(* Logix 5000 project; controller TEC_81 vendor 1 type 14 code 148 rev 36.11; software revision 36.00; part 2 of 4 *)
(* tags used below, declared in another part *)
   Axis_1 : AXIS_CIP_DRIVE;
   Axis_2 : AXIS_CIP_DRIVE;   // Almacen 2
   B_Reset_Posicion_kinetix : DINT;
   Ctrl_Kinetix_A2 : DINT;   // Boton Start Kinetix
   DestornilladorEnPosicion_Mesa : BOOL;   // Sensor de posición de Destornillador en Mesa Central
   Done_Kinetx : DINT;
   Extender_Piston_1_Mesa_Kuka : BOOL;   // Extender Pistón Esquina de Mesa Central
   Extender_Piston_2_Mesa_Kuka : BOOL;   // Extender Pistón Centro de Mesa Central
   Faul_Axis : DINT;
   GripperEnPosicion_Mesa : BOOL;   // Sensor de posición de Gripper en Mesa Central
   In_Pos_Alm_1 : DINT;
   In_Pos_Alm_2 : DINT;
   Kinetix_Pos_Alm_1 : DINT;
   Kinetix_Pos_Alm_2 : DINT;
   KUKA : TIMER;
   MAFR_Mtr_Alm_1 : MOTION_INSTRUCTION;
   MAFR_Mtr_Alm_2 : MOTION_INSTRUCTION;
   MAM_1_Mtr_Alm_0 : MOTION_INSTRUCTION;
   MAM_1_Mtr_Alm_1 : MOTION_INSTRUCTION;
   MAM_1_Mtr_Alm_2 : MOTION_INSTRUCTION;
   MAM_2_Mtr_Alm_1 : MOTION_INSTRUCTION;
   MAM_2_Mtr_Alm_2 : MOTION_INSTRUCTION;
   MAM_3_Mtr_Alm_1 : MOTION_INSTRUCTION;
   MAM_3_Mtr_Alm_2 : MOTION_INSTRUCTION;
   MAM_4_Mtr_Alm_1 : MOTION_INSTRUCTION;
   MAM_4_Mtr_Alm_2 : MOTION_INSTRUCTION;
   MAM_5_Mtr_Alm_1 : MOTION_INSTRUCTION;
   MAM_5_Mtr_Alm_2 : MOTION_INSTRUCTION;
   MAM_6_Mtr_Alm_2 : MOTION_INSTRUCTION;
   ok_com : BOOL;   // tag de prueba de comunicacion
   reset_Kinetix : BOOL;
   Retraer_Piston_1_Mesa_Kuka : BOOL;   // Retraer Pistón Esquina de Mesa Central
   Retraer_Piston_2_Mesa_Kuka : BOOL;   // Retraer Pistón Centro de Mesa Central
   Sensor_Piston_1_Ext_Mesa : BOOL;   // Sensor de Piston Extendido Esquina de la Mesa Central
   Sensor_Piston_1_Ret_Mesa : BOOL;   // Sensor de Pistón Retraido Esquina de la Mesa Central
   Sensor_Piston_2_Ext_Mesa : BOOL;   // Sensor de Pistón Extendido Centro de la Mesa Central
   Sensor_Piston_2_Ret_Mesa : BOOL;   // Sensor de Pistón Retraido Centro de la Mesa Central
   servo_start : MOTION_INSTRUCTION;
   servo_start_01 : MOTION_INSTRUCTION;
   Sevo_Stop : MOTION_INSTRUCTION;
   Start_Kinetix_Alm_1 : DINT;
   Start_Kinetix_Alm_2 : DINT;
   Test : BOOL;
   To_Pos_Alm_1 : DINT;
   To_Pos_Alm_2 : DINT;
   VentosaEnPosicion_Mesa : BOOL;   // Sensor de posición de Ventosa en Mesa Central

PROGRAM _05_Mesa_Central   (* main routine _01_Main *)

ROUTINE _01_Main   (* ladder *)
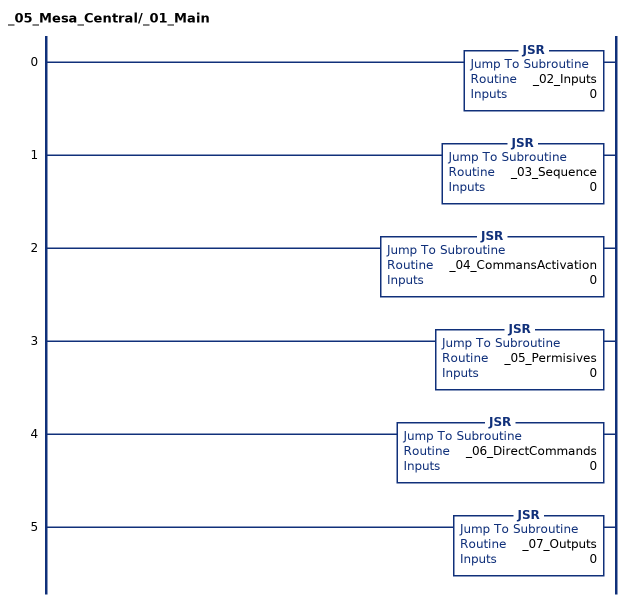
   0: JSR(_02_Inputs,0);
   1: JSR(_03_Sequence,0);
   2: JSR(_04_CommansActivation,0);
   3: JSR(_05_Permisives,0);
   4: JSR(_06_DirectCommands,0);
   5: JSR(_07_Outputs,0);
END_ROUTINE

ROUTINE _02_Inputs   (* ladder *)
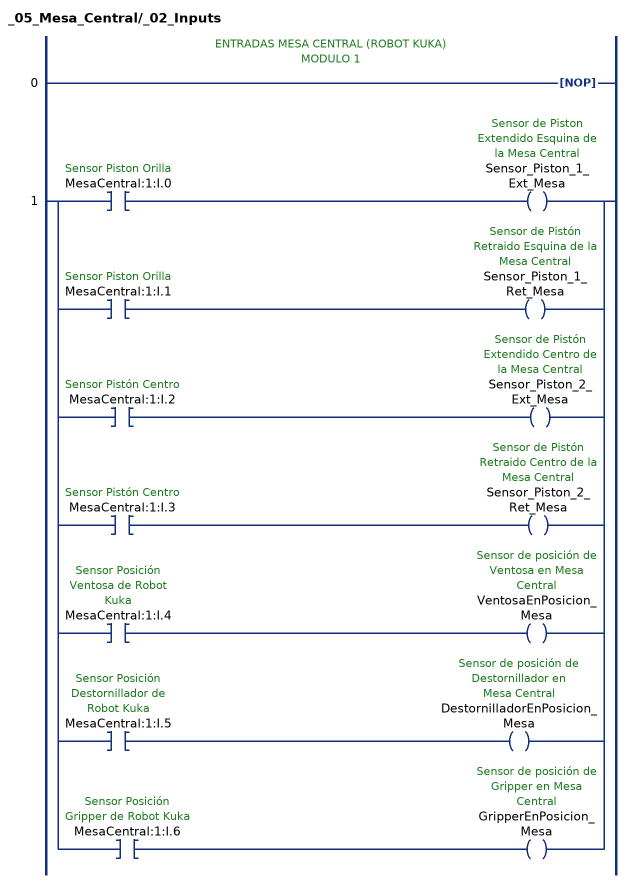
   // ENTRADAS MESA CENTRAL (ROBOT KUKA)
   // MODULO 1
   0: NOP();
   1: [XIC(MesaCentral:1:I.0) OTE(Sensor_Piston_1_Ext_Mesa) ,XIC(MesaCentral:1:I.1) OTE(Sensor_Piston_1_Ret_Mesa) ,XIC(MesaCentral:1:I.2) OTE(Sensor_Piston_2_Ext_Mesa) ,XIC(MesaCentral:1:I.3) OTE(Sensor_Piston_2_Ret_Mesa) ,XIC(MesaCentral:1:I.4) OTE(VentosaEnPosicion_Mesa) ,XIC(MesaCentral:1:I.5) OTE(DestornilladorEnPosicion_Mesa) ,XIC(MesaCentral:1:I.6) OTE(GripperEnPosicion_Mesa) ];
END_ROUTINE

ROUTINE _03_Sequence   (* ladder *)
END_ROUTINE

ROUTINE _04_CommansActivation   (* ladder *)
END_ROUTINE

ROUTINE _05_Permisives   (* ladder *)
END_ROUTINE

ROUTINE _06_DirectCommands   (* ladder *)
END_ROUTINE

ROUTINE _07_Outputs   (* ladder *)
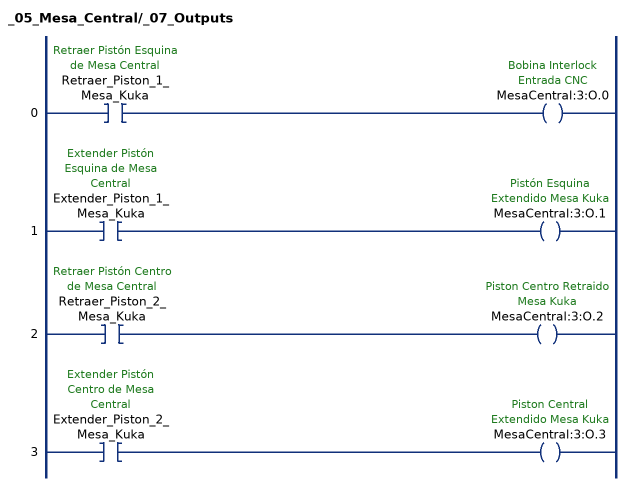
   0: XIC(Retraer_Piston_1_Mesa_Kuka)OTE(MesaCentral:3:O.0);
   1: XIC(Extender_Piston_1_Mesa_Kuka)OTE(MesaCentral:3:O.1);
   2: XIC(Retraer_Piston_2_Mesa_Kuka)OTE(MesaCentral:3:O.2);
   3: XIC(Extender_Piston_2_Mesa_Kuka)OTE(MesaCentral:3:O.3);
END_ROUTINE

ROUTINE test   (* sequential function chart *)
END_ROUTINE

ROUTINE test1   (* ladder *)
END_ROUTINE
END_PROGRAM

PROGRAM _Almacen_1   (* main routine _01_Main_Alm_11 *)
VAR
   B_Reset_Posicion_kinetix_0 : DINT;
   Ctrl_Kinetix_A1 : DINT;
   Done_Kinetx_0 : DINT;
   home_step_1 : BOOL;
   Kinetix_Pos_Alm_0 : DINT;
   ok_com_1 : BOOL;
   reset_Kinetix_1 : BOOL;
END_VAR

ROUTINE _01_Main_Alm_11   (* ladder *)
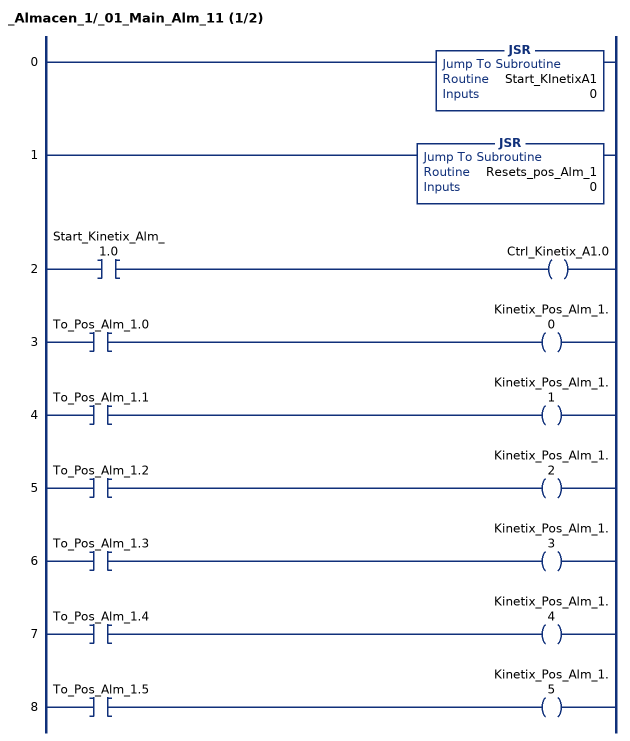
   0: JSR(Start_KInetixA1,0);
   1: JSR(Resets_pos_Alm_1,0);
   2: XIC(Start_Kinetix_Alm_1.0)OTE(Ctrl_Kinetix_A1.0);
   3: XIC(To_Pos_Alm_1.0)OTE(Kinetix_Pos_Alm_1.0);
   4: XIC(To_Pos_Alm_1.1)OTE(Kinetix_Pos_Alm_1.1);
   5: XIC(To_Pos_Alm_1.2)OTE(Kinetix_Pos_Alm_1.2);
   6: XIC(To_Pos_Alm_1.3)OTE(Kinetix_Pos_Alm_1.3);
   7: XIC(To_Pos_Alm_1.4)OTE(Kinetix_Pos_Alm_1.4);
   8: XIC(To_Pos_Alm_1.5)OTE(Kinetix_Pos_Alm_1.5);
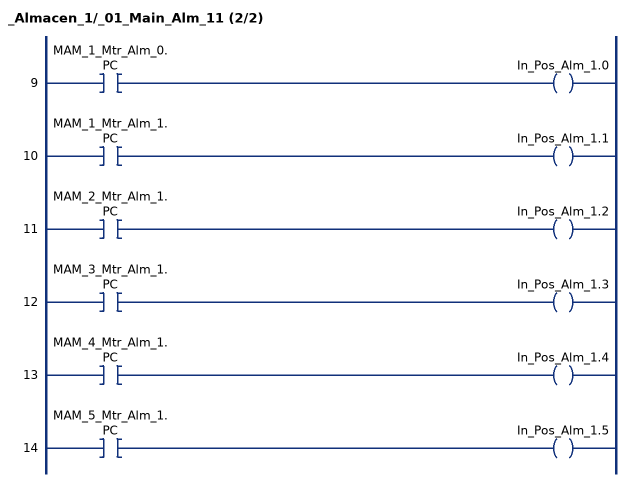
   9: XIC(MAM_1_Mtr_Alm_0.PC)OTE(In_Pos_Alm_1.0);
   10: XIC(MAM_1_Mtr_Alm_1.PC)OTE(In_Pos_Alm_1.1);
   11: XIC(MAM_2_Mtr_Alm_1.PC)OTE(In_Pos_Alm_1.2);
   12: XIC(MAM_3_Mtr_Alm_1.PC)OTE(In_Pos_Alm_1.3);
   13: XIC(MAM_4_Mtr_Alm_1.PC)OTE(In_Pos_Alm_1.4);
   14: XIC(MAM_5_Mtr_Alm_1.PC)OTE(In_Pos_Alm_1.5);
END_ROUTINE

ROUTINE Resets_pos_Alm_1   (* ladder *)
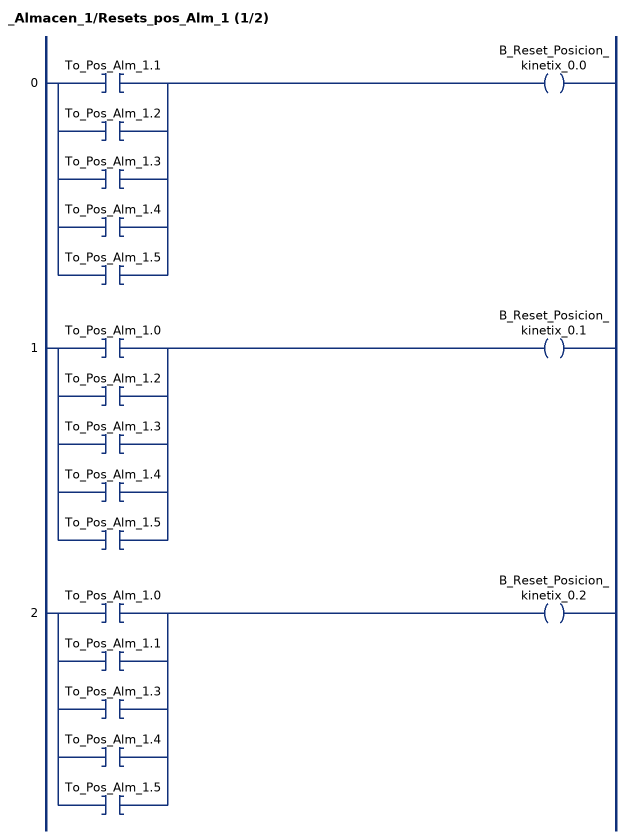
   0: [XIC(To_Pos_Alm_1.1) ,XIC(To_Pos_Alm_1.2) ,XIC(To_Pos_Alm_1.3) ,XIC(To_Pos_Alm_1.4) ,XIC(To_Pos_Alm_1.5) ]OTE(B_Reset_Posicion_kinetix_0.0);
   1: [XIC(To_Pos_Alm_1.0) ,XIC(To_Pos_Alm_1.2) ,XIC(To_Pos_Alm_1.3) ,XIC(To_Pos_Alm_1.4) ,XIC(To_Pos_Alm_1.5) ]OTE(B_Reset_Posicion_kinetix_0.1);
   2: [XIC(To_Pos_Alm_1.0) ,XIC(To_Pos_Alm_1.1) ,XIC(To_Pos_Alm_1.3) ,XIC(To_Pos_Alm_1.4) ,XIC(To_Pos_Alm_1.5) ]OTE(B_Reset_Posicion_kinetix_0.2);
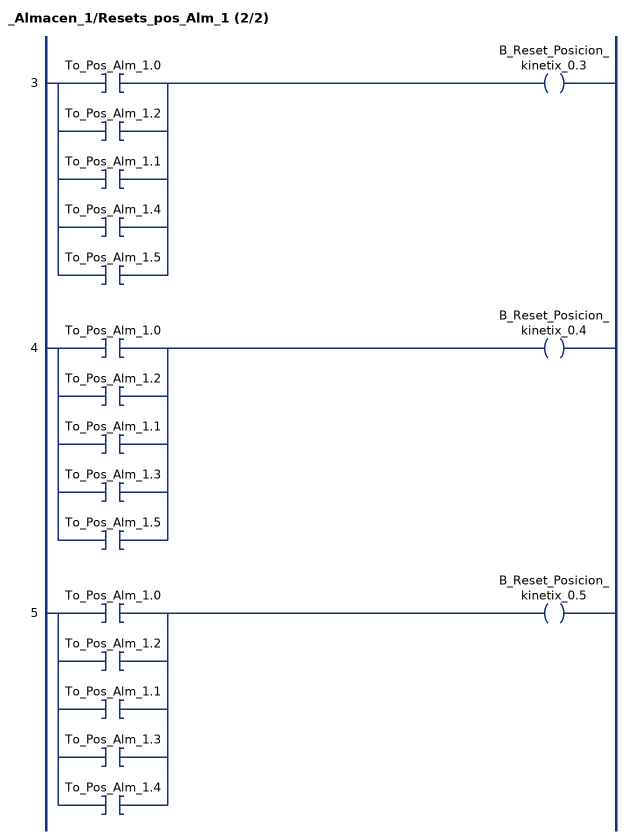
   3: [XIC(To_Pos_Alm_1.0) ,XIC(To_Pos_Alm_1.2) ,XIC(To_Pos_Alm_1.1) ,XIC(To_Pos_Alm_1.4) ,XIC(To_Pos_Alm_1.5) ]OTE(B_Reset_Posicion_kinetix_0.3);
   4: [XIC(To_Pos_Alm_1.0) ,XIC(To_Pos_Alm_1.2) ,XIC(To_Pos_Alm_1.1) ,XIC(To_Pos_Alm_1.3) ,XIC(To_Pos_Alm_1.5) ]OTE(B_Reset_Posicion_kinetix_0.4);
   5: [XIC(To_Pos_Alm_1.0) ,XIC(To_Pos_Alm_1.2) ,XIC(To_Pos_Alm_1.1) ,XIC(To_Pos_Alm_1.3) ,XIC(To_Pos_Alm_1.4) ]OTE(B_Reset_Posicion_kinetix_0.5);
END_ROUTINE

ROUTINE Start_KInetixA1   (* ladder *)
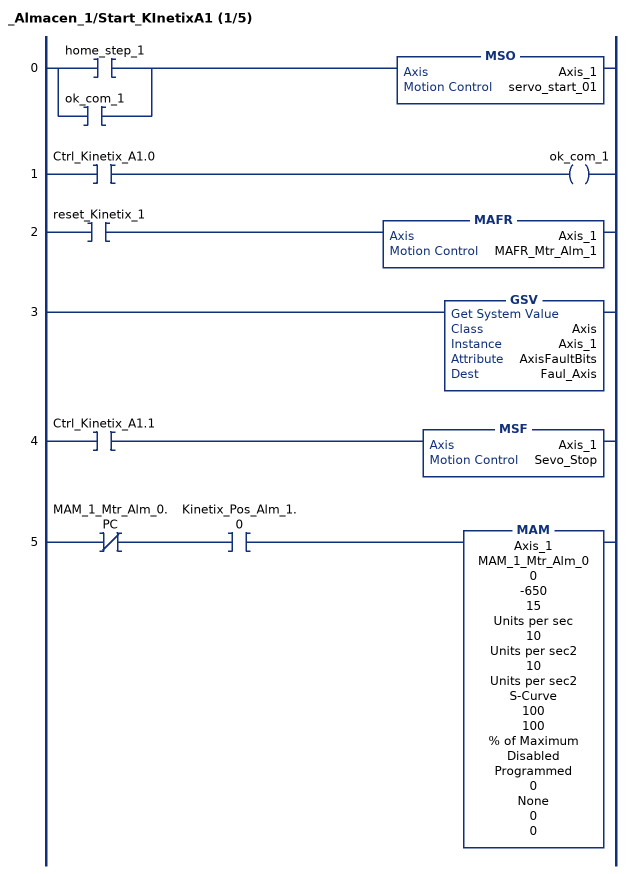
   0: [XIC(home_step_1) ,XIC(ok_com_1) ]MSO(Axis_1,servo_start_01);
   1: XIC(Ctrl_Kinetix_A1.0)OTE(ok_com_1);
   2: XIC(reset_Kinetix_1)MAFR(Axis_1,MAFR_Mtr_Alm_1);
   3: GSV(Axis,Axis_1,AxisFaultBits,Faul_Axis);
   4: XIC(Ctrl_Kinetix_A1.1)MSF(Axis_1,Sevo_Stop);
   5: XIO(MAM_1_Mtr_Alm_0.PC)XIC(Kinetix_Pos_Alm_1.0)MAM(Axis_1,MAM_1_Mtr_Alm_0,0,-650,15,Units per sec,10,Units per sec2,10,Units per sec2,S-Curve,100,100,% of Maximum,Disabled,Programmed,0,None,0,0);
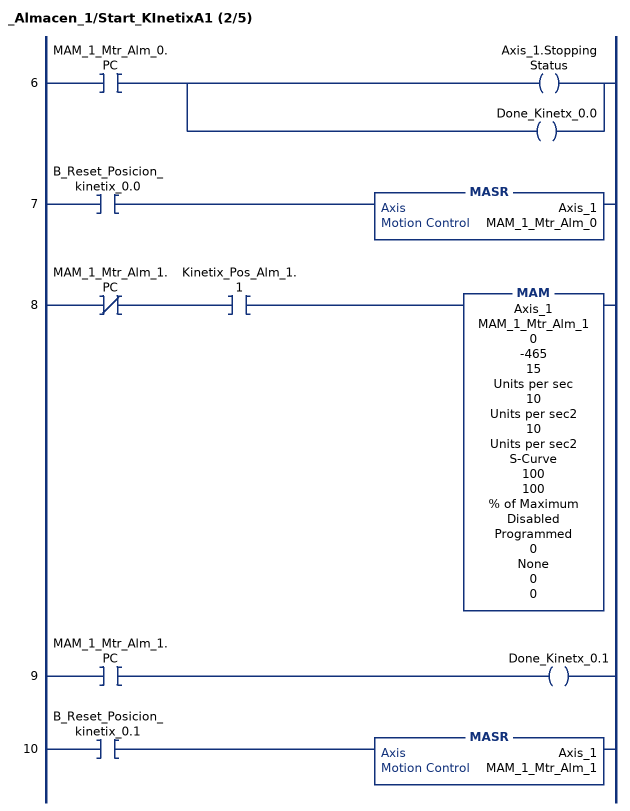
   6: XIC(MAM_1_Mtr_Alm_0.PC)[OTE(Axis_1.StoppingStatus) ,OTE(Done_Kinetx_0.0) ];
   7: XIC(B_Reset_Posicion_kinetix_0.0)MASR(Axis_1,MAM_1_Mtr_Alm_0);
   8: XIO(MAM_1_Mtr_Alm_1.PC)XIC(Kinetix_Pos_Alm_1.1)MAM(Axis_1,MAM_1_Mtr_Alm_1,0,-465,15,Units per sec,10,Units per sec2,10,Units per sec2,S-Curve,100,100,% of Maximum,Disabled,Programmed,0,None,0,0);
   9: XIC(MAM_1_Mtr_Alm_1.PC)OTE(Done_Kinetx_0.1);
   10: XIC(B_Reset_Posicion_kinetix_0.1)MASR(Axis_1,MAM_1_Mtr_Alm_1);
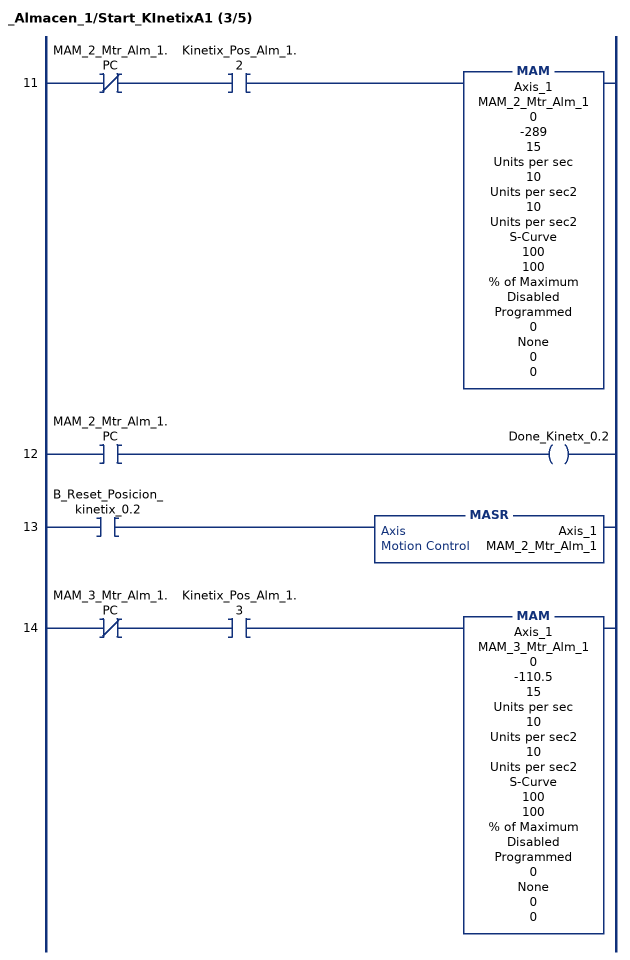
   11: XIO(MAM_2_Mtr_Alm_1.PC)XIC(Kinetix_Pos_Alm_1.2)MAM(Axis_1,MAM_2_Mtr_Alm_1,0,-289,15,Units per sec,10,Units per sec2,10,Units per sec2,S-Curve,100,100,% of Maximum,Disabled,Programmed,0,None,0,0);
   12: XIC(MAM_2_Mtr_Alm_1.PC)OTE(Done_Kinetx_0.2);
   13: XIC(B_Reset_Posicion_kinetix_0.2)MASR(Axis_1,MAM_2_Mtr_Alm_1);
   14: XIO(MAM_3_Mtr_Alm_1.PC)XIC(Kinetix_Pos_Alm_1.3)MAM(Axis_1,MAM_3_Mtr_Alm_1,0,-110.5,15,Units per sec,10,Units per sec2,10,Units per sec2,S-Curve,100,100,% of Maximum,Disabled,Programmed,0,None,0,0);
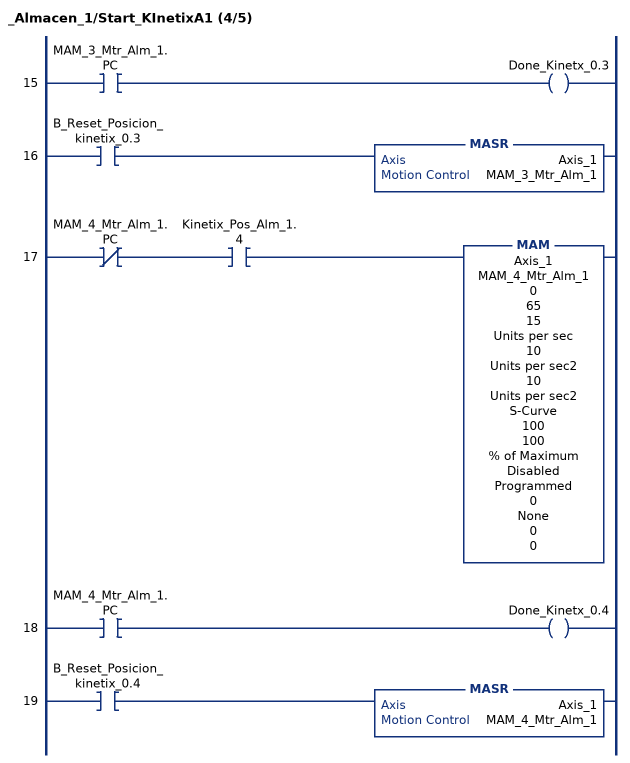
   15: XIC(MAM_3_Mtr_Alm_1.PC)OTE(Done_Kinetx_0.3);
   16: XIC(B_Reset_Posicion_kinetix_0.3)MASR(Axis_1,MAM_3_Mtr_Alm_1);
   17: XIO(MAM_4_Mtr_Alm_1.PC)XIC(Kinetix_Pos_Alm_1.4)MAM(Axis_1,MAM_4_Mtr_Alm_1,0,65,15,Units per sec,10,Units per sec2,10,Units per sec2,S-Curve,100,100,% of Maximum,Disabled,Programmed,0,None,0,0);
   18: XIC(MAM_4_Mtr_Alm_1.PC)OTE(Done_Kinetx_0.4);
   19: XIC(B_Reset_Posicion_kinetix_0.4)MASR(Axis_1,MAM_4_Mtr_Alm_1);
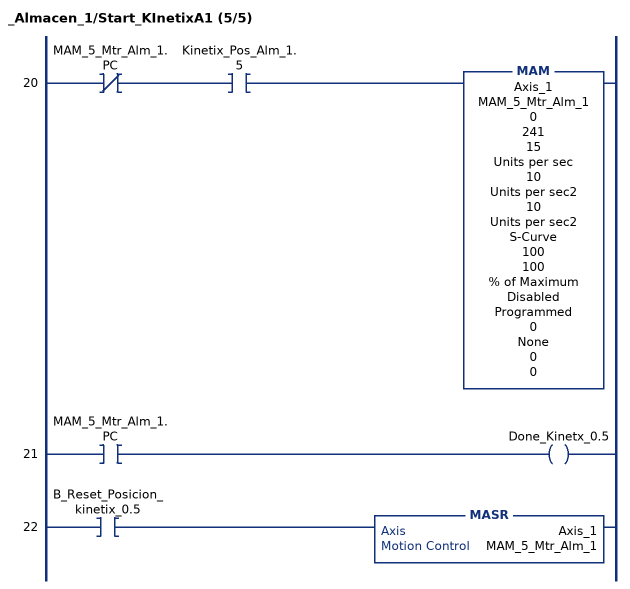
   20: XIO(MAM_5_Mtr_Alm_1.PC)XIC(Kinetix_Pos_Alm_1.5)MAM(Axis_1,MAM_5_Mtr_Alm_1,0,241,15,Units per sec,10,Units per sec2,10,Units per sec2,S-Curve,100,100,% of Maximum,Disabled,Programmed,0,None,0,0);
   21: XIC(MAM_5_Mtr_Alm_1.PC)OTE(Done_Kinetx_0.5);
   22: XIC(B_Reset_Posicion_kinetix_0.5)MASR(Axis_1,MAM_5_Mtr_Alm_1);
END_ROUTINE
END_PROGRAM

PROGRAM _Almacen_2   (* main routine _01_Main *)
VAR
   home_step : BOOL;
END_VAR

ROUTINE _01_Main   (* ladder *)
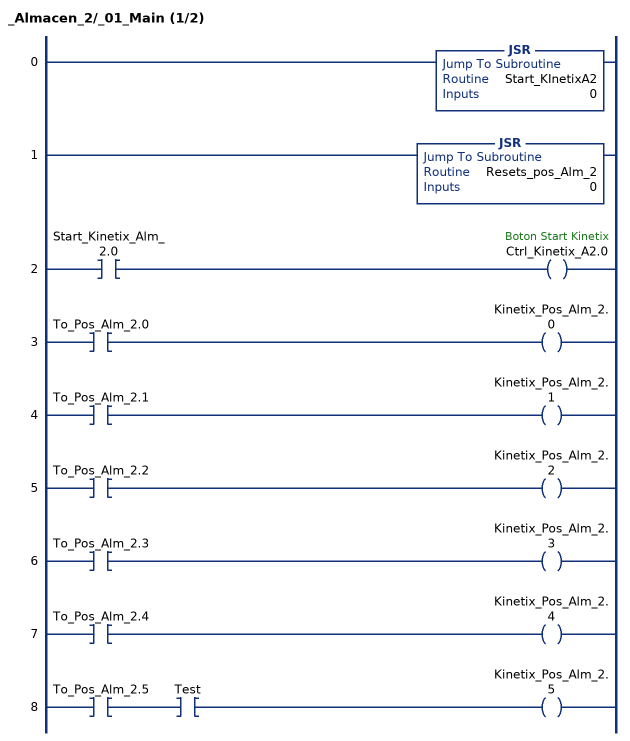
   0: JSR(Start_KInetixA2,0);
   1: JSR(Resets_pos_Alm_2,0);
   2: XIC(Start_Kinetix_Alm_2.0)OTE(Ctrl_Kinetix_A2.0);
   3: XIC(To_Pos_Alm_2.0)OTE(Kinetix_Pos_Alm_2.0);
   4: XIC(To_Pos_Alm_2.1)OTE(Kinetix_Pos_Alm_2.1);
   5: XIC(To_Pos_Alm_2.2)OTE(Kinetix_Pos_Alm_2.2);
   6: XIC(To_Pos_Alm_2.3)OTE(Kinetix_Pos_Alm_2.3);
   7: XIC(To_Pos_Alm_2.4)OTE(Kinetix_Pos_Alm_2.4);
   8: XIC(To_Pos_Alm_2.5)XIC(Test)OTE(Kinetix_Pos_Alm_2.5);
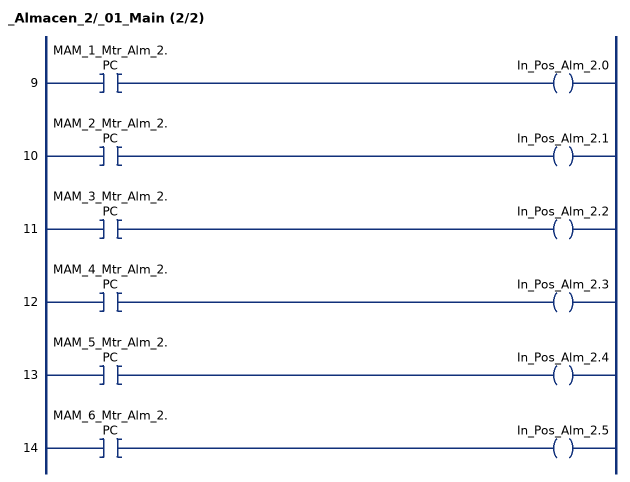
   9: XIC(MAM_1_Mtr_Alm_2.PC)OTE(In_Pos_Alm_2.0);
   10: XIC(MAM_2_Mtr_Alm_2.PC)OTE(In_Pos_Alm_2.1);
   11: XIC(MAM_3_Mtr_Alm_2.PC)OTE(In_Pos_Alm_2.2);
   12: XIC(MAM_4_Mtr_Alm_2.PC)OTE(In_Pos_Alm_2.3);
   13: XIC(MAM_5_Mtr_Alm_2.PC)OTE(In_Pos_Alm_2.4);
   14: XIC(MAM_6_Mtr_Alm_2.PC)OTE(In_Pos_Alm_2.5);
END_ROUTINE

ROUTINE Resets_pos_Alm_2   (* ladder *)
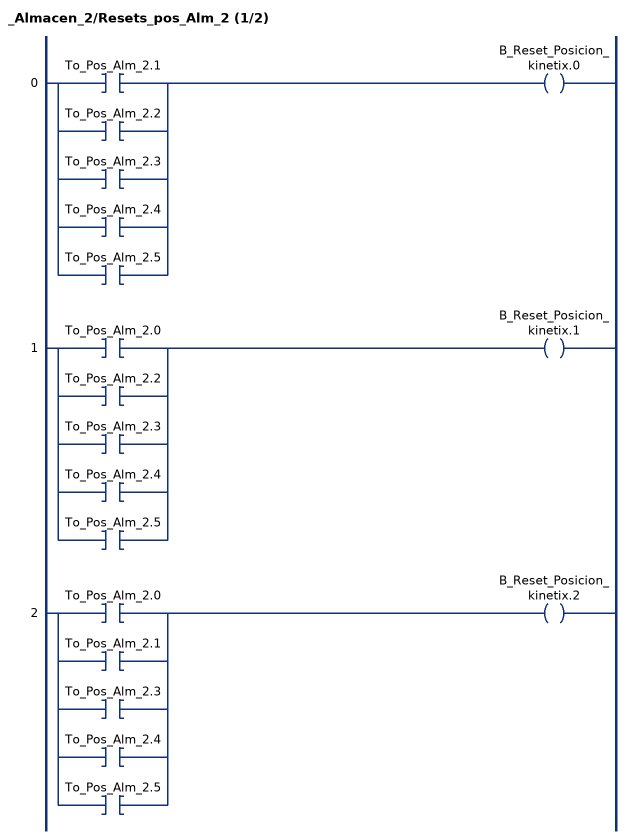
   0: [XIC(To_Pos_Alm_2.1) ,XIC(To_Pos_Alm_2.2) ,XIC(To_Pos_Alm_2.3) ,XIC(To_Pos_Alm_2.4) ,XIC(To_Pos_Alm_2.5) ]OTE(B_Reset_Posicion_kinetix.0);
   1: [XIC(To_Pos_Alm_2.0) ,XIC(To_Pos_Alm_2.2) ,XIC(To_Pos_Alm_2.3) ,XIC(To_Pos_Alm_2.4) ,XIC(To_Pos_Alm_2.5) ]OTE(B_Reset_Posicion_kinetix.1);
   2: [XIC(To_Pos_Alm_2.0) ,XIC(To_Pos_Alm_2.1) ,XIC(To_Pos_Alm_2.3) ,XIC(To_Pos_Alm_2.4) ,XIC(To_Pos_Alm_2.5) ]OTE(B_Reset_Posicion_kinetix.2);
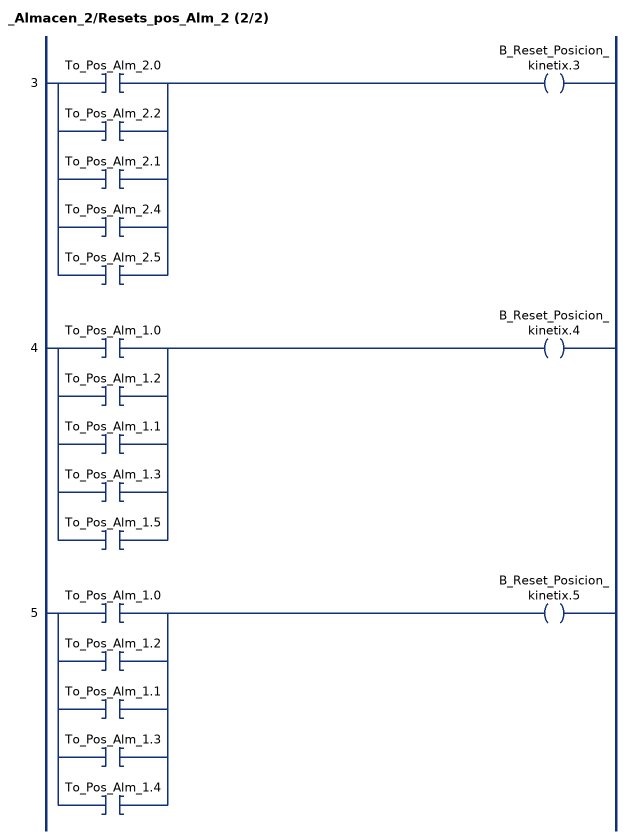
   3: [XIC(To_Pos_Alm_2.0) ,XIC(To_Pos_Alm_2.2) ,XIC(To_Pos_Alm_2.1) ,XIC(To_Pos_Alm_2.4) ,XIC(To_Pos_Alm_2.5) ]OTE(B_Reset_Posicion_kinetix.3);
   4: [XIC(To_Pos_Alm_1.0) ,XIC(To_Pos_Alm_1.2) ,XIC(To_Pos_Alm_1.1) ,XIC(To_Pos_Alm_1.3) ,XIC(To_Pos_Alm_1.5) ]OTE(B_Reset_Posicion_kinetix.4);
   5: [XIC(To_Pos_Alm_1.0) ,XIC(To_Pos_Alm_1.2) ,XIC(To_Pos_Alm_1.1) ,XIC(To_Pos_Alm_1.3) ,XIC(To_Pos_Alm_1.4) ]OTE(B_Reset_Posicion_kinetix.5);
END_ROUTINE

ROUTINE Start_KInetixA2   (* ladder *)
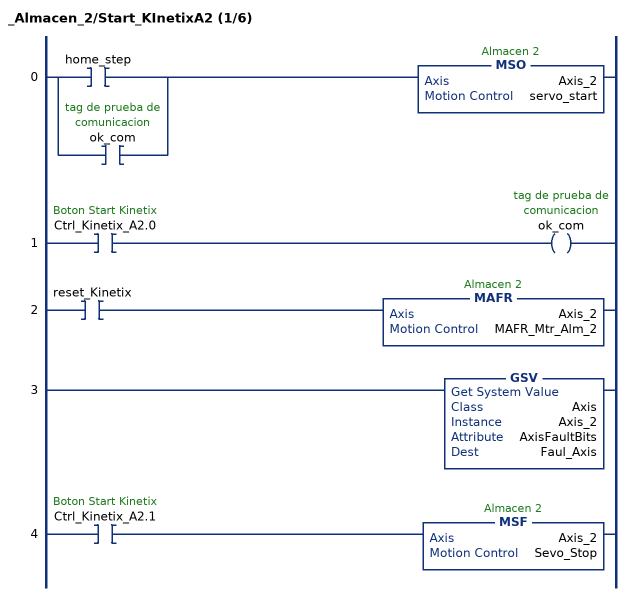
   0: [XIC(home_step) ,XIC(ok_com) ]MSO(Axis_2,servo_start);
   1: XIC(Ctrl_Kinetix_A2.0)OTE(ok_com);
   2: XIC(reset_Kinetix)MAFR(Axis_2,MAFR_Mtr_Alm_2);
   3: GSV(Axis,Axis_2,AxisFaultBits,Faul_Axis);
   4: XIC(Ctrl_Kinetix_A2.1)MSF(Axis_2,Sevo_Stop);
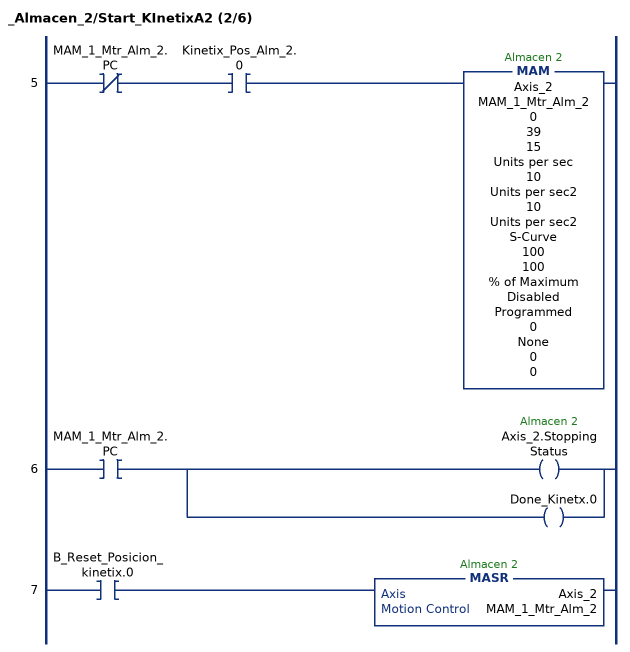
   5: XIO(MAM_1_Mtr_Alm_2.PC)XIC(Kinetix_Pos_Alm_2.0)MAM(Axis_2,MAM_1_Mtr_Alm_2,0,39,15,Units per sec,10,Units per sec2,10,Units per sec2,S-Curve,100,100,% of Maximum,Disabled,Programmed,0,None,0,0);
   6: XIC(MAM_1_Mtr_Alm_2.PC)[OTE(Axis_2.StoppingStatus) ,OTE(Done_Kinetx.0) ];
   7: XIC(B_Reset_Posicion_kinetix.0)MASR(Axis_2,MAM_1_Mtr_Alm_2);
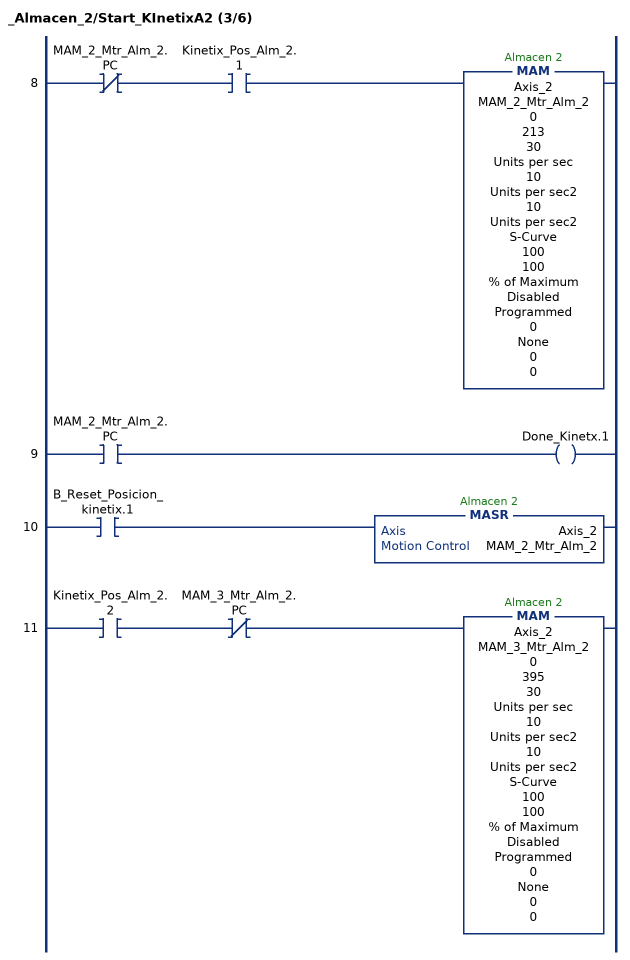
   8: XIO(MAM_2_Mtr_Alm_2.PC)XIC(Kinetix_Pos_Alm_2.1)MAM(Axis_2,MAM_2_Mtr_Alm_2,0,213,30,Units per sec,10,Units per sec2,10,Units per sec2,S-Curve,100,100,% of Maximum,Disabled,Programmed,0,None,0,0);
   9: XIC(MAM_2_Mtr_Alm_2.PC)OTE(Done_Kinetx.1);
   10: XIC(B_Reset_Posicion_kinetix.1)MASR(Axis_2,MAM_2_Mtr_Alm_2);
   11: XIC(Kinetix_Pos_Alm_2.2)XIO(MAM_3_Mtr_Alm_2.PC)MAM(Axis_2,MAM_3_Mtr_Alm_2,0,395,30,Units per sec,10,Units per sec2,10,Units per sec2,S-Curve,100,100,% of Maximum,Disabled,Programmed,0,None,0,0);
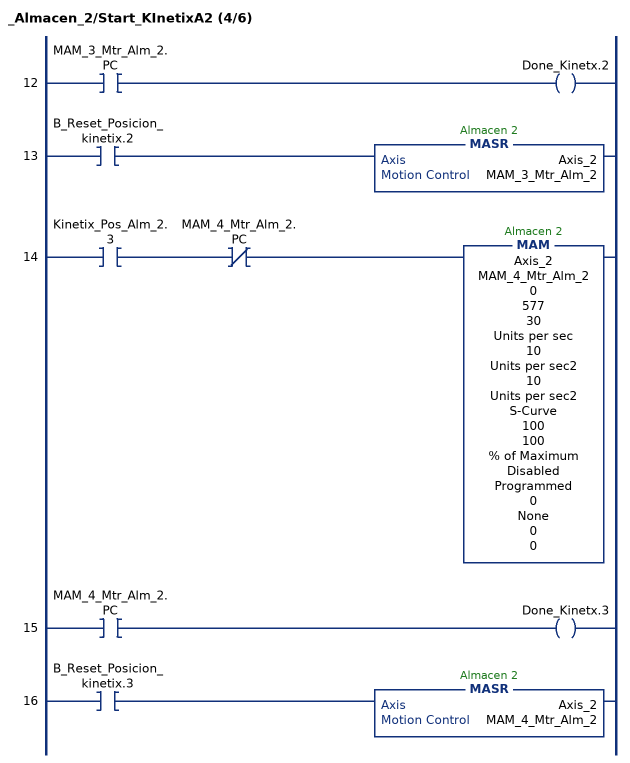
   12: XIC(MAM_3_Mtr_Alm_2.PC)OTE(Done_Kinetx.2);
   13: XIC(B_Reset_Posicion_kinetix.2)MASR(Axis_2,MAM_3_Mtr_Alm_2);
   14: XIC(Kinetix_Pos_Alm_2.3)XIO(MAM_4_Mtr_Alm_2.PC)MAM(Axis_2,MAM_4_Mtr_Alm_2,0,577,30,Units per sec,10,Units per sec2,10,Units per sec2,S-Curve,100,100,% of Maximum,Disabled,Programmed,0,None,0,0);
   15: XIC(MAM_4_Mtr_Alm_2.PC)OTE(Done_Kinetx.3);
   16: XIC(B_Reset_Posicion_kinetix.3)MASR(Axis_2,MAM_4_Mtr_Alm_2);
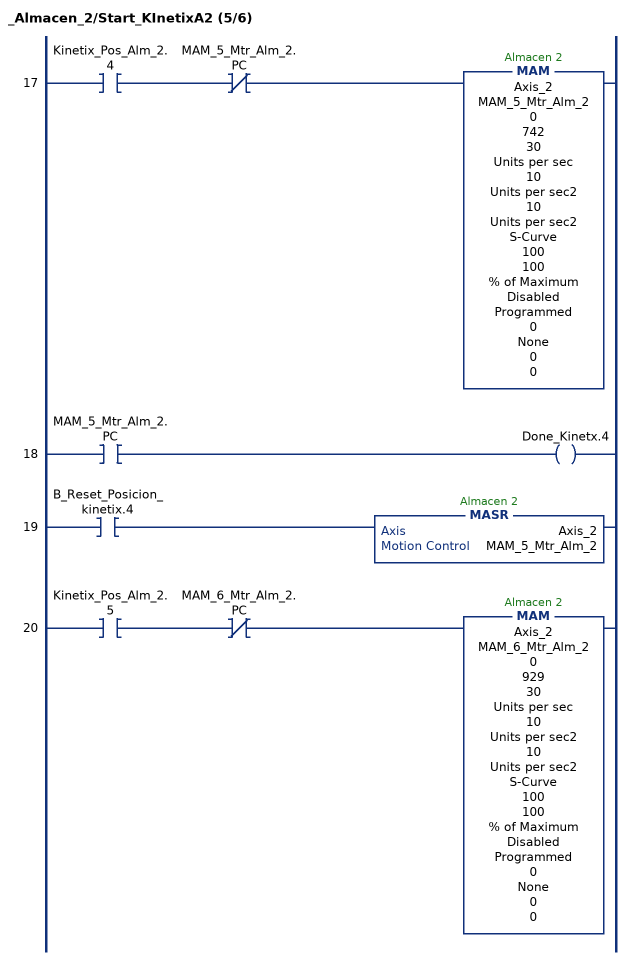
   17: XIC(Kinetix_Pos_Alm_2.4)XIO(MAM_5_Mtr_Alm_2.PC)MAM(Axis_2,MAM_5_Mtr_Alm_2,0,742,30,Units per sec,10,Units per sec2,10,Units per sec2,S-Curve,100,100,% of Maximum,Disabled,Programmed,0,None,0,0);
   18: XIC(MAM_5_Mtr_Alm_2.PC)OTE(Done_Kinetx.4);
   19: XIC(B_Reset_Posicion_kinetix.4)MASR(Axis_2,MAM_5_Mtr_Alm_2);
   20: XIC(Kinetix_Pos_Alm_2.5)XIO(MAM_6_Mtr_Alm_2.PC)MAM(Axis_2,MAM_6_Mtr_Alm_2,0,929,30,Units per sec,10,Units per sec2,10,Units per sec2,S-Curve,100,100,% of Maximum,Disabled,Programmed,0,None,0,0);
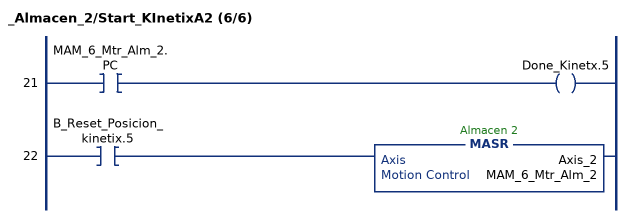
   21: XIC(MAM_6_Mtr_Alm_2.PC)OTE(Done_Kinetx.5);
   22: XIC(B_Reset_Posicion_kinetix.5)MASR(Axis_2,MAM_6_Mtr_Alm_2);
END_ROUTINE
END_PROGRAM
